Fanuc TP program (LS listing): a_calw1.ls

/PROG  A_CALW1
/ATTR
OWNER		= MNEDITOR;
COMMENT		= "";
PROG_SIZE	= 5497;
CREATE		= DATE 13-09-16  TIME 12:40:42;
MODIFIED	= DATE 18-03-07  TIME 13:07:56;
FILE_NAME	= AUTO_CAL;
VERSION		= 0;
LINE_COUNT	= 300;
MEMORY_SIZE	= 5961;
PROTECT		= READ_WRITE;
TCD:  STACK_SIZE	= 0,
      TASK_PRIORITY	= 50,
      TIME_SLICE	= 0,
      BUSY_LAMP_OFF	= 0,
      ABORT_REQUEST	= 0,
      PAUSE_REQUEST	= 0;
DEFAULT_GROUP	= 1,*,*,*,*;
CONTROL_CODE	= 00000000 00000000;
/APPL
  ARC : TRUE ;
  ARC Welding Equipment : 1,*,*,*,*;

MPAS ;
MPAS_NUM_PASSES        : 0;
MPAS_LAST_PASS         : 0;
MPAS_CURRENT_PASS      : 0;
MPAS_STATUS_PASS       : 0;
/MN
   1:  !****************************** ;
   2:  !**** WIRE CALIBRATION ;
   :!****  25 deg angle *******;
   3:  !****************************** ;
   4:  OVERRIDE=100% ;
   5:   ;
   6:  !If Robot is not folded ;
   7:  PR[120]=JPOS    ;
   8:  IF (PR[120,2]<70) THEN ;
   9:  CALL FOLD1    ;
  10:  ENDIF ;
  11:   ;
  12:  !------- SENS OVERRIDE ------- ;
  13:  R[135]=50    ;
  14:   ;
  15:  UTOOL_NUM=9 ;
  16:  UFRAME_NUM=8 ;
  17:   ;
  18:  !------- TOOL WIDTH ------- ;
  19:   ;
  20:   ;
  21:  !------- SET ZERO TOOL ------- ;
  22:  PR[180]=LPOS    ;
  23:  PR[180,1]=0    ;
  24:  PR[180,2]=0    ;
  25:  PR[180,3]=0    ;
  26:  PR[180,4]=0    ;
  27:  PR[180,5]=0    ;
  28:  PR[180,6]=0    ;
  29:   ;
  30:  UTOOL[9]=PR[180] ;
  31:   ;
  32:  ! to get correct userframe ;
  33:  PR[180,6]=90    ;
  34:  UFRAME[8]=PR[180] ;
  35:  PR[180,6]=0    ;
  36:   ;
  37:  !Touch sensing off ;
  38:  DO[256]=OFF ;
  39:   ;
  40:   ;
  41:  PR[126]=LPOS    ;
  42:  IF (PR[126,1]>550),JMP LBL[120] ;
  43:  PR[126,1]=PR[126,1]+100    ;
  44:   ;
  45:L PR[126] 50mm/sec FINE    ;
  46:   ;
  47:  !------- UNFOLD POINT ------- ;
  48:  LBL[120] ;
  49:  PR[120]=JPOS    ;
  50:  PR[120,1]=90    ;
  51:  PR[120,7]=1000    ;
  52:J PR[120] 50% FINE    ;
  53:   ;
  54:  LBL[121] ;
  55:  PR[121]=JPOS    ;
  56:  PR[121,1]=90    ;
  57:  PR[121,2]=90    ;
  58:  PR[121,3]=(-80)    ;
  59:  PR[121,4]=0    ;
  60:  PR[121,5]=30    ;
  61:  PR[121,6]=0    ;
  62:   ;
  63:J PR[121] 50% FINE    ;
  64:   ;
  65:  PR[122]=PR[121]    ;
  66:  PR[122,5]=(-100)    ;
  67:J PR[122] 50% FINE    ;
  68:   ;
  69:   ;
  70:  !****************************** ;
  71:  !**** SENSING ;
  72:  !****************************** ;
  73:   ;
  74:  !------------ Z1 --------------- ;
  75:   ;
  76:  PR[124]=LPOS    ;
  77:  PR[124,1]=485    ;
  78:  PR[124,2]=PR[124,2]    ;
  79:  PR[124,3]=(-415)    ;
  80:  PR[124,4]=0    ;
  81:  PR[124,5]=90    ;
  82:  PR[124,6]=180    ;
  83:   ;
  84:L PR[124] 50mm/sec FINE    ;
  85:   ;
  86:  PR[160]=PR[124]    ;
  87:  PR[160,1]=PR[160,1]-40    ;
  88:  SKIP CONDITION DI[256]=ON    ;
  89:   ;
  90:  OVERRIDE=R[135] ;
  91:  DO[256]=ON ;
  92:L PR[160] 1mm/sec FINE Skip,LBL[991],PR[170]=LPOS    ;
  93:   ;
  94:  DO[256]=OFF ;
  95:  OVERRIDE=100% ;
  96:   ;
  97:  !****************************** ;
  98:  !------------ X1 --------------- ;
  99:   ;
 100:L PR[124] 50mm/sec FINE    ;
 101:   ;
 102:  PR[125]=PR[124]    ;
 103:  PR[125,2]=PR[125,2]-100    ;
 104:  PR[125,3]=(-480)    ;
 105:L PR[125] 50mm/sec FINE    ;
 106:   ;
 107:   ;
 108:  PR[123]=PR[124]    ;
 109:  PR[123,1]=PR[170,1]-5    ;
 110:  PR[123,2]=PR[123,2]-90    ;
 111:  PR[123,3]=(-350)    ;
 112:  PR[123,4]=90    ;
 113:  PR[123,5]=0    ;
 114:  PR[123,6]=(-90)    ;
 115:   ;
 116:L PR[123] 50mm/sec FINE    ;
 117:   ;
 118:  PR[161]=PR[123]    ;
 119:  PR[161,2]=PR[161,2]+40    ;
 120:  SKIP CONDITION DI[256]=ON    ;
 121:   ;
 122:  OVERRIDE=R[135] ;
 123:  DO[256]=ON ;
 124:L PR[161] 1mm/sec FINE Skip,LBL[991],PR[171]=LPOS    ;
 125:   ;
 126:  DO[256]=OFF ;
 127:  OVERRIDE=100% ;
 128:   ;
 129:  !------------ X2 --------------- ;
 130:   ;
 131:L PR[123] 50mm/sec FINE    ;
 132:   ;
 133:  PR[125]=LPOS    ;
 134:  PR[125,1]=PR[125,1]+20    ;
 135:L PR[125] 50mm/sec FINE    ;
 136:L PR[124] 48mm/sec FINE    ;
 137:   ;
 138:  PR[125]=PR[124]    ;
 139:  PR[125,2]=PR[125,2]+100    ;
 140:  PR[125,3]=(-480)    ;
 141:L PR[125] 50mm/sec FINE    ;
 142:   ;
 143:  PR[126]=PR[123]    ;
 144:  PR[126,2]=PR[124,2]+90    ;
 145:  PR[126,4]=PR[123,4]*(-1)    ;
 146:  PR[126,5]=0    ;
 147:  PR[126,6]=PR[123,6]*(-1)    ;
 148:   ;
 149:L PR[126] 50mm/sec FINE    ;
 150:   ;
 151:  PR[162]=PR[126]    ;
 152:  PR[162,2]=PR[162,2]-40    ;
 153:  SKIP CONDITION DI[256]=ON    ;
 154:   ;
 155:  OVERRIDE=R[135] ;
 156:  DO[256]=ON ;
 157:L PR[162] 1mm/sec FINE Skip,LBL[991],PR[172]=LPOS    ;
 158:   ;
 159:  DO[256]=OFF ;
 160:  OVERRIDE=100% ;
 161:   ;
 162:  PR[180,1]=(((PR[172,2]-PR[171,2]-30)/2-.5)*(-1)) ;
 163:   ;
 164:  !****************************** ;
 165:  !------------ Y1 --------------- ;
 166:   ;
 167:L PR[126] 48mm/sec FINE    ;
 168:  PR[125]=LPOS    ;
 169:  PR[125,1]=PR[125,1]+20    ;
 170:L PR[125] 50mm/sec FINE    ;
 171:L PR[124] 50mm/sec FINE    ;
 172:   ;
 173:  PR[123]=LPOS    ;
 174:  PR[123,1]=PR[170,1]-5    ;
 175:  PR[123,2]=PR[124,2]-70    ;
 176:  PR[123,3]=(-365)    ;
 177:  PR[123,4]=90    ;
 178:  PR[123,5]=0    ;
 179:  PR[123,6]=(-90)    ;
 180:   ;
 181:  PR[125]=PR[124]    ;
 182:  PR[125,1]=PR[125,1]+50    ;
 183:  PR[125,3]=PR[125,3]-50    ;
 184:L PR[125] 50mm/sec FINE    ;
 185:L PR[123] 50mm/sec FINE    ;
 186:   ;
 187:  PR[163]=PR[123]    ;
 188:  PR[163,3]=PR[163,3]+40    ;
 189:  SKIP CONDITION DI[256]=ON    ;
 190:   ;
 191:  OVERRIDE=R[135] ;
 192:  DO[256]=ON ;
 193:L PR[163] 1mm/sec FINE Skip,LBL[991],PR[173]=LPOS    ;
 194:   ;
 195:  DO[256]=OFF ;
 196:  OVERRIDE=100% ;
 197:   ;
 198:  !------------ Y2 --------------- ;
 199:   ;
 200:L PR[123] 125mm/sec CNT50    ;
 201:L PR[125] 60mm/sec FINE    ;
 202:   ;
 203:  PR[126]=PR[123]    ;
 204:  PR[126,2]=PR[124,2]+70    ;
 205:  PR[126,4]=(-90)    ;
 206:  PR[126,6]=90    ;
 207:   ;
 208:L PR[126] 50mm/sec FINE    ;
 209:   ;
 210:  PR[164]=PR[126]    ;
 211:  PR[164,3]=PR[164,3]+40    ;
 212:  SKIP CONDITION DI[256]=ON    ;
 213:   ;
 214:  OVERRIDE=R[135] ;
 215:  DO[256]=ON ;
 216:L PR[164] 1mm/sec FINE Skip,LBL[991],PR[174]=LPOS    ;
 217:   ;
 218:  DO[256]=OFF ;
 219:  OVERRIDE=100% ;
 220:   ;
 221:  PR[180,2]=((PR[174,3]-PR[173,3])/2) ;
 222:   ;
 223:  !****************************** ;
 224:  !------------ Z2 --------------- ;
 225:   ;
 226:  PR[126,1]=500    ;
 227:L PR[126] 125mm/sec CNT50    ;
 228:   ;
 229:  PR[127]=LPOS    ;
 230:  PR[127,1]=275    ;
 231:  PR[127,2]=PR[124,2]-67    ;
 232:  PR[127,3]=(-32)    ;
 233:  PR[127,4]=(-180)    ;
 234:  PR[127,5]=0    ;
 235:  PR[127,6]=0    ;
 236:   ;
 237:  PR[125]=PR[127]    ;
 238:  PR[125,1]=500    ;
 239:  PR[125,2]=PR[124,2]    ;
 240:L PR[125] 60mm/sec FINE    ;
 241:   ;
 242:L PR[127] 120mm/sec FINE    ;
 243:   ;
 244:  PR[165]=PR[127]    ;
 245:  PR[165,3]=PR[165,3]-40    ;
 246:  SKIP CONDITION DI[256]=ON    ;
 247:   ;
 248:  OVERRIDE=R[135] ;
 249:  DO[256]=ON ;
 250:L PR[165] 1mm/sec FINE Skip,LBL[991],PR[175]=LPOS    ;
 251:   ;
 252:  DO[256]=OFF ;
 253:  OVERRIDE=100% ;
 254:   ;
 255:   ;
 256:  PR[180,3]=(PR[175,3]-PR[174,3]+PR[180,2]-25-.5) ;
 257:   ;
 258:   ;
 259:  !****************************** ;
 260:  !**** SET TOOL POINT ;
 261:  !****************************** ;
 262:   ;
 263:   ;
 264:  !----- ;
 265:  PR[180,4]=(-180)    ;
 266:  PR[180,5]=(-25)    ;
 267:  PR[180,6]=0    ;
 268:   ;
 269:  UTOOL[1]=PR[180] ;
 270:   ;
 271:L PR[125] 60mm/sec FINE    ;
 272:J PR[121] 50% CNT50    ;
 273:   ;
 274:  JMP LBL[9999] ;
 275:   ;
 276:  !****************************** ;
 277:  !**** ERROR HANDLING ;
 278:  !****************************** ;
 279:  LBL[991] ;
 280:  DO[256]=OFF ;
 281:  R[162]=603    ;
 282:   ;
 283:  PR[126]=LPOS    ;
 284:  PR[126,1]=PR[126,1]+100    ;
 285:   ;
 286:L PR[126] 50mm/sec FINE    ;
 287:   ;
 288:J PR[121] 50% FINE    ;
 289:  ABORT ;
 290:   ;
 291:  LBL[9999] ;
 292:  OVERRIDE=100% ;
 293:  CALL FOLD1    ;
 294:  UTOOL_NUM=1 ;
 295:  UFRAME_NUM=1 ;
 296:  !Calibration OK ;
 297:  R[215]=6070    ;
 298:   ;
 299:   ;
 300:   ;
/POS
/END
